# B&R Automation Studio project Teknologia25 (part 4)

#### Types.typ - Exported data types
```iecst
TYPE
	brfiShuttleSelectionType : 	STRUCT
		ID : DINT;
		index : DINT;
		x : REAL;
		y : REAL;
	END_STRUCT;
END_TYPE

(**)
(*----- brfi6DMoveQueue -----*)

TYPE
	brfi6DMoveQueueStateEnum :
		(
		brfi6DMOVEQUEUE_DISABLED,
		brfi6DMOVEQUEUE_RUN,
		brfi6DMOVEQUEUE_DONE,
		brfi6DMOVEQUEUE_ERROR
		);
	brfi6DMoveQueueFbType : 	STRUCT
		ShGetInfo : MC_BR_ShGetInfo_Acp6D;
		MoveInPlane : MC_BR_MoveInPlane_Acp6D;
		Move6D : MC_BR_Move6D_Acp6D;
		MoveArc : MC_BR_MoveArc_Acp6D;
		ShWaitTime : MC_BR_ShWaitTime_Acp6D;
		RotaryMotion : MC_BR_RotaryMotion_Acp6D;
		ShLevitation : MC_BR_ShLevitation_Acp6D;
		RotaryMotionSpin : MC_BR_RotaryMotionSpin_Acp6D;
		ShWaitCmdLb : MC_BR_ShWaitCmdLb_Acp6D;
	END_STRUCT;
	brfi6DMoveQueueIrnalType : 	STRUCT
		initialized : BOOL;
		onStateEntry : BOOL;
		lastState : brfi6DMoveQueueStateEnum;
		lastSubState : DINT;
		i : DINT;
		position : McAcp6DShPositionType;
		Xc : REAL;
		Yc : REAL;
		dx : REAL;
		dy : REAL;
		radius : REAL;
		angle : REAL;
	END_STRUCT;
	brfi6DMoveQueueActionsType : 	STRUCT
		acknowledge : BOOL;
		error : BOOL;
		done : BOOL;
		getInfo : BOOL;
	END_STRUCT;
	brfi6DMoveQueueExecuteType : 	STRUCT
		moveInPlane : BOOL;
		move6D : BOOL;
		moveArc : BOOL;
		wait : BOOL;
		moveRotary : BOOL;
		levitate : BOOL;
		spin : BOOL;
		readInfo : BOOL;
		waitCmdLb : BOOL;
	END_STRUCT;
	brfi6DMoveQueueCommandType : 	STRUCT
		mask : UINT;
		inPlane : McAcp6DInPlaneParType;
		inSpace : McAcp6DMove6DParType;
		moveMode6D : McAcp6DMoveModeEnum;
		waitTime : REAL;
		rotary : McAcp6DRotaryMotionParType;
		arc : McAcp6DArcParType;
		levitation : McAcp6DLevitationParType;
		spin : McAcp6DRotaryMotionSpinParType;
		waitCmdLb : brfi6DMoveWaitLabelParamType;
	END_STRUCT;
	brfi6DMoveQueueParamType : 	STRUCT
		velocity_xy : REAL;
		velocity_short : REAL;
		velocity_rotary : REAL;
		acceleration : REAL;
		acceleration_rotary : REAL;
	END_STRUCT;
	brfi6DMoveCommandSelectionEnum :
		(
		sX := 1,
		sY := 2,
		sZ := 4,
		sRx := 8,
		sRy := 16,
		sRz := 32,
		sArc := 64,
		sRotary := 128,
		sWait := 256,
		sLevitate := 512,
		sSpin := 1024,
		sUpdatePosition := 2048,
		sWaitCmdLb := 4096
		);
	brfi6DMoveCommandPathEnum :
		(
		pathDIRECT,
		pathX_Y,
		pathY_X
		);
	brfi6DMoveWaitLabelParamType : 	STRUCT
		monitoredShuttleID : UINT;
		triggerType : McAcp6DShWaitCmdLbTriggerEnum;
		commandLabel : UINT;
		labelType : McAcp6DShWaitCmdLbLabelEnum;
	END_STRUCT;
END_TYPE

(**)

TYPE
	Acp6dShuttleType : 	STRUCT  (*Global shuttle list datatype*)
		ID : UINT; (*ID of the shuttle*)
		Ref : Mc6DShuttleType; (*Reference to the shuttle*)
		index : DINT; (*ID of the shuttle*)
		status : Acp6dShuttleStatusType; (*Reference to the shuttle*)
		position : Acp6dShuttlePositionType;
		force : Acp6dShuttleForceType;
		command : Acp6dShuttleCmdType;
		moveCyclicActive : BOOL;
	END_STRUCT;
	Acp6dShuttleCmdType : 	STRUCT  (*Global shuttle list datatype*)
		move6D : BOOL; (*ID of the shuttle*)
		moveQueue : BOOL; (*ID of the shuttle*)
	END_STRUCT;
	Acp6dShuttlePositionType : 	STRUCT  (*Global shuttle list datatype*)
		isValid : BOOL; (*ID of the shuttle*)
		value : McAcp6DShPositionType; (*ID of the shuttle*)
	END_STRUCT;
	Acp6dShuttleForceType : 	STRUCT  (*Global shuttle list datatype*)
		isValid : BOOL; (*ID of the shuttle*)
		value : McAcp6DShForceType; (*ID of the shuttle*)
		Z_avg : REAL;
		Fz_baseline : REAL;
		readings : ARRAY[0..gMAX_INDEX_MEASUREMENT]OF McAcp6DShForceType;
	END_STRUCT;
	Acp6dShuttleStatusType : 	STRUCT  (*Global shuttle list datatype*)
		isValid : BOOL; (*ID of the shuttle*)
		state : McAcp6DShStateEnum; (*ID of the shuttle*)
	END_STRUCT;
END_TYPE

(**)

TYPE
	brfiShuttleGroupFbType : 	STRUCT
		GroupCreate : MC_BR_ShGroupCreate_Acp6D;
		GroupAddShuttle : MC_BR_ShGroupAddShuttle_Acp6D;
		GroupDelete : MC_BR_ShGroupDelete_Acp6D;
		GroupGetInfo : MC_BR_ShGroupGetInfo_Acp6D;
		GroupCoupleCtrl : MC_BR_ShGroupCoupleCtrl_Acp6D;
	END_STRUCT;
END_TYPE

(**)
```

#### Constants.var - Exported constants
```iecst
VAR CONSTANT
	MEASUREMENT_COUNT : DINT := 10;
	MAX_NUM_SHUTTLE : DINT := 8; (*Maximum numer of shuttles on the system*)
	MAX_NUM_SHUTTLE_VIRTUAL : DINT := 2; (*Maximum numer of shuttles on the system*)
	MAX_NUM_TARGETS : DINT := 20; (*Maximum numer of shuttles on the system*)
	SHUFFLE_SEQUENCE_LEN : DINT := 16;
END_VAR
(**)
VAR CONSTANT
	gMAX_INDEX_SHUTTLE : DINT := MAX_NUM_SHUTTLE - 1; (*Maximum index for a shuttles on the system*)
	gMAX_INDEX_SHUTTLE_VIRTUAL : DINT := MAX_NUM_SHUTTLE_VIRTUAL - 1; (*Maximum index for a shuttles on the system*)
	gMAX_INDEX_TARGETS : DINT := MAX_NUM_TARGETS - 1; (*Maximum index for a shuttles on the system*)
	gMAX_INDEX_MEASUREMENT : DINT := MEASUREMENT_COUNT - 1;
	gMAX_INDEX_SHUFFLE : DINT := SHUFFLE_SEQUENCE_LEN - 1;
END_VAR
(**)
```

#### brfiDemo.fun - Exported functions and function blocks
```iecst
{REDUND_ERROR} FUNCTION brfiShuffle : BOOL (* *) (*$GROUP=User,$CAT=User,$GROUPICON=User.png,$CATICON=User.png*)
	VAR_INPUT
		refArray : REFERENCE TO ARRAY[0..gMAX_INDEX_SHUTTLE] OF DINT;
	END_VAR
	VAR
		newOrder : ARRAY[0..gMAX_INDEX_SHUTTLE] OF DINT;
		added : ARRAY[0..gMAX_INDEX_SHUTTLE] OF BOOL;
		rand : DINT;
		count : DINT;
		i : DINT;
		ordinal : DINT;
		x : DINT;
	END_VAR
END_FUNCTION

FUNCTION brfiShuttleSelect : DINT
	VAR_INPUT
		Shuttles : REFERENCE TO ARRAY[0..gMAX_INDEX_SHUTTLE] OF Acp6dShuttleType;
		Selection : REFERENCE TO ARRAY[0..gMAX_INDEX_SHUTTLE] OF brfiShuttleSelectionType;
		X0 : REAL;
		Y0 : REAL;
		X1 : REAL;
		Y1 : REAL;
	END_VAR
	VAR
		i : DINT;
		j : DINT;
		count : DINT;
		maxX : REAL;
		maxY : REAL;
		minX : REAL;
		minY : REAL;
		key : brfiShuttleSelectionType;
	END_VAR
END_FUNCTION

FUNCTION brfiShuttleSelectClosest : DINT
	VAR_INPUT
		Shuttles : REFERENCE TO ARRAY[0..gMAX_INDEX_SHUTTLE] OF Acp6dShuttleType;
		X : REAL;
		Y : REAL;
	END_VAR
	VAR
		i : DINT;
		dist : REAL;
		dist_min : REAL;
		index_min : DINT;
	END_VAR
END_FUNCTION

FUNCTION brfiSortCompare : BOOL
	VAR_INPUT
		A : brfiShuttleSelectionType;
		B : brfiShuttleSelectionType;
		AscendingX : BOOL;
		AscendingY : BOOL;
	END_VAR
	VAR
		isEqualX : BOOL;
	END_VAR
END_FUNCTION

FUNCTION brfiToRAD : REAL
	VAR_INPUT
		degrees : REAL;
	END_VAR
END_FUNCTION

FUNCTION brfiToDEG : REAL
	VAR_INPUT
		radians : REAL;
	END_VAR
END_FUNCTION
(**)

{REDUND_ERROR} FUNCTION_BLOCK brfi6DMoveQueue (* *) (*$GROUP=User,$CAT=User,$GROUPICON=User.png,$CATICON=User.png*)
	VAR_INPUT
		Shuttle : REFERENCE TO Mc6DShuttleType;
		Execute : {REDUND_UNREPLICABLE} BOOL;
		Parameters : {REDUND_UNREPLICABLE} brfi6DMoveQueueParamType;
		Commands : {REDUND_UNREPLICABLE} ARRAY[0..gMAX_INDEX_TARGETS] OF brfi6DMoveQueueCommandType;
	END_VAR
	VAR_OUTPUT
		Done : {REDUND_UNREPLICABLE} BOOL;
		Acknowledge : {REDUND_UNREPLICABLE} BOOL;
		Error : {REDUND_UNREPLICABLE} BOOL;
		ErrorID : {REDUND_UNREPLICABLE} DINT;
		FailedCommand : {REDUND_UNREPLICABLE} brfi6DMoveQueueCommandType;
		FailedCommandIndex : {REDUND_UNREPLICABLE} DINT;
		LastExecutedState : {REDUND_UNREPLICABLE} DINT;
	END_VAR
	VAR
		refCommand : REFERENCE TO brfi6DMoveQueueCommandType;
		refAllCommandsDone : REFERENCE TO BOOL;
		state : {REDUND_UNREPLICABLE} brfi6DMoveQueueStateEnum;
		subState : {REDUND_UNREPLICABLE} DINT;
		onStateEntry : BOOL;
		fb : {REDUND_UNREPLICABLE} brfi6DMoveQueueFbType;
		actions : {REDUND_UNREPLICABLE} brfi6DMoveQueueActionsType;
		cmd : {REDUND_UNREPLICABLE} brfi6DMoveQueueExecuteType;
		internal : {REDUND_UNREPLICABLE} brfi6DMoveQueueIrnalType;
	END_VAR
END_FUNCTION_BLOCK

FUNCTION AddCommand6D_xy : BOOL
	VAR_INPUT
		Commands : REFERENCE TO ARRAY[0..gMAX_INDEX_TARGETS] OF brfi6DMoveQueueCommandType;
		axisSelect : brfi6DMoveCommandSelectionEnum;
		x : REAL;
		y : REAL;
		velocity : REAL;
		acceleration : REAL;
		endVelocity : REAL;
		path : brfi6DMoveCommandPathEnum;
		radius : REAL;
		mode : McAcp6DMoveModeEnum;
	END_VAR
	VAR
		i : DINT;
	END_VAR
END_FUNCTION

FUNCTION AddCommand6D_xyz : BOOL
	VAR_INPUT
		Commands : REFERENCE TO ARRAY[0..gMAX_INDEX_TARGETS] OF brfi6DMoveQueueCommandType;
		axisSelect : brfi6DMoveCommandSelectionEnum;
		x : REAL;
		y : REAL;
		z : REAL;
		velocity : REAL;
		velocity_short : REAL;
		acceleration : REAL;
		mode : McAcp6DMoveModeEnum;
	END_VAR
	VAR
		i : DINT;
	END_VAR
END_FUNCTION

FUNCTION AddCommand6D_Rxyz : BOOL
	VAR_INPUT
		Commands : REFERENCE TO ARRAY[0..gMAX_INDEX_TARGETS] OF brfi6DMoveQueueCommandType;
		axisSelect : brfi6DMoveCommandSelectionEnum;
		Rx : REAL;
		Ry : REAL;
		Rz : REAL;
		velocity_short : REAL;
		mode : McAcp6DMoveModeEnum;
	END_VAR
	VAR
		i : DINT;
	END_VAR
END_FUNCTION

FUNCTION AddCommand6D_wait : BOOL
	VAR_INPUT
		Commands : REFERENCE TO ARRAY[0..gMAX_INDEX_TARGETS] OF brfi6DMoveQueueCommandType;
		time : REAL; (*wait time in seconds*)
	END_VAR
	VAR
		i : DINT;
	END_VAR
END_FUNCTION

FUNCTION AddCommand6D_land : BOOL
	VAR_INPUT
		Commands : REFERENCE TO ARRAY[0..gMAX_INDEX_TARGETS] OF brfi6DMoveQueueCommandType;
		speed : USINT;
		Fz : REAL;
	END_VAR
	VAR
		i : DINT;
	END_VAR
END_FUNCTION

FUNCTION AddCommand6D_levitate : BOOL
	VAR_INPUT
		Commands : REFERENCE TO ARRAY[0..gMAX_INDEX_TARGETS] OF brfi6DMoveQueueCommandType;
		speed : USINT;
		Fz : REAL;
	END_VAR
	VAR
		i : DINT;
	END_VAR
END_FUNCTION

FUNCTION AddCommand6D_spin : BOOL
	VAR_INPUT
		Commands : REFERENCE TO ARRAY[0..gMAX_INDEX_TARGETS] OF brfi6DMoveQueueCommandType;
		duration : REAL; (*Duration of the rotational movement after reaching the target velocity (s)*)
		angle : REAL; (*Angle at which the shuttle stops after the rotational movement (rad)*)
		velocity : REAL; (*Rotational speed (rad/s)*)
		acceleration : REAL; (*Rotational acceleration (rad/s2)*)
	END_VAR
	VAR
		i : DINT;
	END_VAR
END_FUNCTION

FUNCTION AddCommand6D_rotateAbs : BOOL
	VAR_INPUT
		Commands : REFERENCE TO ARRAY[0..gMAX_INDEX_TARGETS] OF brfi6DMoveQueueCommandType;
		angle : REAL; (*Target angle (rad)*)
		velocity : REAL; (*Rotational speed (rad/s)*)
		acceleration : REAL; (*Rotational acceleration (rad/s2)*)
	END_VAR
	VAR
		i : DINT;
	END_VAR
END_FUNCTION

FUNCTION AddCommand6D_rotateCW : BOOL
	VAR_INPUT
		Commands : REFERENCE TO ARRAY[0..gMAX_INDEX_TARGETS] OF brfi6DMoveQueueCommandType;
		angle : REAL; (*Target angle (rad)*)
		velocity : REAL; (*Rotational speed (rad/s)*)
		acceleration : REAL; (*Rotational acceleration (rad/s2)*)
	END_VAR
	VAR
		i : DINT;
	END_VAR
END_FUNCTION

FUNCTION AddCommand6D_rotateCCW : BOOL
	VAR_INPUT
		Commands : REFERENCE TO ARRAY[0..gMAX_INDEX_TARGETS] OF brfi6DMoveQueueCommandType;
		angle : REAL; (*Target angle (rad)*)
		velocity : REAL; (*Rotational speed (rad/s)*)
		acceleration : REAL; (*Rotational acceleration (rad/s2)*)
	END_VAR
	VAR
		i : DINT;
	END_VAR
END_FUNCTION

FUNCTION AddCommand6D_arcAngularCW : BOOL
	VAR_INPUT
		Commands : REFERENCE TO ARRAY[0..gMAX_INDEX_TARGETS] OF brfi6DMoveQueueCommandType;
		x : REAL;
		y : REAL;
		angle : REAL;
		velocity : REAL;
		acceleration : REAL;
		endVelocity : REAL;
		mode : McAcp6DMoveModeEnum;
	END_VAR
	VAR
		i : DINT;
	END_VAR
END_FUNCTION

FUNCTION AddCommand6D_arcAngularCCW : BOOL
	VAR_INPUT
		Commands : REFERENCE TO ARRAY[0..gMAX_INDEX_TARGETS] OF brfi6DMoveQueueCommandType;
		x : REAL;
		y : REAL;
		angle : REAL;
		velocity : REAL;
		acceleration : REAL;
		endVelocity : REAL;
		mode : McAcp6DMoveModeEnum;
	END_VAR
	VAR
		i : DINT;
	END_VAR
END_FUNCTION

FUNCTION AddCommand6D_arcRadialCW : BOOL
	VAR_INPUT
		Commands : REFERENCE TO ARRAY[0..gMAX_INDEX_TARGETS] OF brfi6DMoveQueueCommandType;
		x : REAL;
		y : REAL;
		radius : REAL;
		type : McAcp6DArcTypeEnum; (*Rotational speed (rad/s)*)
		velocity : REAL; (*Rotational speed (rad/s)*)
		acceleration : REAL; (*Rotational acceleration (rad/s2)*)
		endVelocity : REAL; (*Target angle (rad)*)
		mode : McAcp6DMoveModeEnum;
	END_VAR
	VAR
		i : DINT;
	END_VAR
END_FUNCTION

FUNCTION AddCommand6D_arcRadialCCW : BOOL
	VAR_INPUT
		Commands : REFERENCE TO ARRAY[0..gMAX_INDEX_TARGETS] OF brfi6DMoveQueueCommandType;
		x : REAL;
		y : REAL;
		radius : REAL;
		type : McAcp6DArcTypeEnum; (*Rotational speed (rad/s)*)
		velocity : REAL; (*Rotational speed (rad/s)*)
		acceleration : REAL; (*Rotational acceleration (rad/s2)*)
		endVelocity : REAL; (*Target angle (rad)*)
		mode : McAcp6DMoveModeEnum;
	END_VAR
	VAR
		i : DINT;
	END_VAR
END_FUNCTION

FUNCTION AddCommand6D_waitCmdLb : BOOL
	VAR_INPUT
		Commands : REFERENCE TO ARRAY[0..gMAX_INDEX_TARGETS] OF brfi6DMoveQueueCommandType;
		monitoredShuttleID : UINT;
		triggerType : McAcp6DShWaitCmdLbTriggerEnum;
		commandLabel : UINT;
		labelType : McAcp6DShWaitCmdLbLabelEnum;
	END_VAR
	VAR
		i : DINT;
	END_VAR
END_FUNCTION
(**)

{REDUND_ERROR} FUNCTION_BLOCK brfiShuttleGroup (* *) (*$GROUP=User,$CAT=User,$GROUPICON=User.png,$CATICON=User.png*)
	VAR_INPUT
		Assembly : REFERENCE TO Mc6DAssemblyType;
		Shuttles : {REDUND_UNREPLICABLE} ARRAY[0..gMAX_INDEX_SHUTTLE] OF Mc6DShuttleType;
		Enable : {REDUND_UNREPLICABLE} BOOL;
	END_VAR
	VAR_OUTPUT
		Inactive : {REDUND_UNREPLICABLE} BOOL;
		Active : {REDUND_UNREPLICABLE} BOOL;
		Busy : {REDUND_UNREPLICABLE} BOOL;
		Error : {REDUND_UNREPLICABLE} BOOL;
		ErrorID : {REDUND_UNREPLICABLE} DINT;
		NumberOfShuttles : {REDUND_UNREPLICABLE} UINT;
	END_VAR
	VAR
		shuttleGroupRef : Mc6DShuttleGroupType;
		state : {REDUND_UNREPLICABLE} DINT;
		i : {REDUND_UNREPLICABLE} DINT;
		fb : {REDUND_UNREPLICABLE} brfiShuttleGroupFbType;
	END_VAR
END_FUNCTION_BLOCK
(**)

{REDUND_ERROR} FUNCTION_BLOCK brfiSunPlanet (* *) (*$GROUP=User,$CAT=User,$GROUPICON=User.png,$CATICON=User.png*)
	VAR_INPUT
		SunShuttle : REFERENCE TO Mc6DShuttleType;
		PlanetShuttles : {REDUND_UNREPLICABLE} ARRAY[0..gMAX_INDEX_SHUTTLE] OF Mc6DShuttleType;
		Enable : {REDUND_UNREPLICABLE} BOOL;
	END_VAR
	VAR_OUTPUT
		Active : {REDUND_UNREPLICABLE} BOOL;
		Busy : {REDUND_UNREPLICABLE} BOOL;
		Error : {REDUND_UNREPLICABLE} BOOL;
		ErrorID : {REDUND_UNREPLICABLE} DINT;
	END_VAR
	VAR
		state : {REDUND_UNREPLICABLE} DINT;
		i : {REDUND_UNREPLICABLE} DINT;
		ShPlanet : {REDUND_UNREPLICABLE} MC_BR_ShPlanet_Acp6D;
	END_VAR
END_FUNCTION_BLOCK
```

#### Common.st
```iecst
(*  *)
FUNCTION brfiShuffle

	count := gMAX_INDEX_SHUTTLE;

	FOR i := 0 TO gMAX_INDEX_SHUTTLE DO
		rand := RandValueDINT(0, count);
		ordinal := 0;

		FOR x := 0 TO gMAX_INDEX_SHUTTLE DO
			IF NOT added[x] THEN
				ordinal := ordinal + 1;
			END_IF;

			IF (rand + 1) = ordinal THEN
				EXIT;
			END_IF;
		END_FOR;

		added[x] := TRUE;
		newOrder[x] := refArray[i];
		count := count - 1;

	END_FOR;

	brsmemcpy(ADR(refArray), ADR(newOrder), SIZEOF(refArray));

END_FUNCTION

FUNCTION brfiShuttleSelect

	// First find shuttles that are in the selection area
	maxX := MAX(X0, X1);
	maxY := MAX(Y0, Y1);
	minX := MIN(X0, X1);
	minY := MIN(Y0, Y1);
	brsmemset(ADR(Selection), 0, SIZEOF(Selection));

	FOR i := 0 TO gMAX_INDEX_SHUTTLE DO
		IF Shuttles[i].position.value.X < maxX AND Shuttles[i].position.value.X > minX THEN
			IF Shuttles[i].position.value.Y < maxY AND Shuttles[i].position.value.Y > minY THEN
				Selection[count].index := Shuttles[i].index;
				Selection[count].ID := Shuttles[i].ID;
				Selection[count].x := Shuttles[i].position.value.X;
				Selection[count].y := Shuttles[i].position.value.Y;
				count := count + 1;
			END_IF;
		END_IF;
	END_FOR;

	brfiShuttleSelect := count;

	IF count < 2 THEN
		RETURN;
	END_IF;

	// Sort selection array by X
	FOR i := 1 TO count - 1 DO
		key := Selection[i];
		j := i - 1;

		// Compare key with each element on the LEFT OF it UNTIL an element smaller than it is found
		WHILE j >= 0 AND brfiSortCompare(key, Selection[j], (X0 < X1), (Y0 < Y1)) DO
			Selection[j + 1] := Selection[j];
			j := j - 1;
			Selection[j + 1] := key;
		END_WHILE;
	END_FOR

END_FUNCTION

FUNCTION brfiShuttleSelectClosest

	dist_min := 1000000;

	FOR i := 0 TO gMAX_INDEX_SHUTTLE DO
		dist := SQRT(EXPT(X - Shuttles[i].position.value.X, 2) + EXPT(Y - Shuttles[i].position.value.Y, 2));

		IF  dist < dist_min THEN
			dist_min := dist;
	  		index_min := i;
		END_IF;
	END_FOR;

	brfiShuttleSelectClosest := index_min;

END_FUNCTION

FUNCTION brfiSortCompare
	// Comparison function for two pairs (A, B)

	IF AscendingX THEN
		// X needs to be sorted in ascending order
		IF A.x < B.x THEN
			brfiSortCompare := TRUE;
			RETURN;
		END_IF;
	ELSE
		// X needs to be sorted in descending order
		IF A.x > B.x THEN
			brfiSortCompare := TRUE;
			RETURN;
		END_IF;
	END_IF;

	isEqualX := ABS(A.x - B.x) < 0.001;

	IF isEqualX THEN
		// Only sort by Y if X is equal as we primarily sort by X
		IF AscendingY THEN
			// Y needs to be sorted in ascending order
			IF A.y < B.y THEN
				brfiSortCompare := TRUE;
				RETURN;
			END_IF;
		ELSE
			// Y needs to be sorted in descending order
			IF A.y > B.y THEN
				brfiSortCompare := TRUE;
				RETURN;
			END_IF;
		END_IF;
	END_IF;

END_FUNCTION

FUNCTION brfiToRAD

	brfiToRAD := degrees * brmPI / 180.0;

END_FUNCTION

FUNCTION brfiToDEG

	brfiToDEG := radians / brmPI * 180.0;

END_FUNCTION
```

#### MoveQueue.st
```iecst
FUNCTION_BLOCK brfi6DMoveQueue

    // Execution control
    // ========================================================================================================
	IF Execute = FALSE THEN
		IF internal.initialized THEN
			brsmemset(ADR(internal), 0, SIZEOF(internal));
			brsmemset(ADR(actions), 0, SIZEOF(actions));
		END_IF
		state := brfi6DMOVEQUEUE_DISABLED;
	END_IF

	// Program code
	// ========================================================================================================
	CASE state OF
		brfi6DMOVEQUEUE_DISABLED:
			//
			// ------------------------------------------------------
			IF Execute THEN
				internal.initialized := TRUE;
				brsmemset(ADR(FailedCommand), 0, SIZEOF(FailedCommand));
				brsmemset(ADR(cmd), 0, SIZEOF(cmd));
				FailedCommandIndex := -1;
				ErrorID := 0;
				state := brfi6DMOVEQUEUE_RUN;
			END_IF;

		brfi6DMOVEQUEUE_RUN:
			CASE subState OF
				0:
					// ------------------------------------------------------
					actions.getInfo := TRUE;

					IF fb.ShGetInfo.Done THEN
						internal.position := fb.ShGetInfo.ShuttleInfo.Position;
						subState := 100;
					ELSIF fb.ShGetInfo.Error THEN
						ErrorID := fb.ShGetInfo.ErrorID;
						state := brfi6DMOVEQUEUE_ERROR;
					END_IF;

				100:
					// Find next target that has masked axes
					// ------------------------------------------------------
					IF internal.i > gMAX_INDEX_TARGETS THEN
						state := brfi6DMOVEQUEUE_DONE;
					END_IF;

					WHILE internal.i <= gMAX_INDEX_TARGETS DO
						refCommand ACCESS ADR(Commands[internal.i]);

						IF refCommand.mask > 0 THEN
							// Select movement type based on the AxisMask for the target
							IF refCommand.mask <= 3 THEN
								cmd.moveInPlane := FALSE;
								subState := 200;
	  						ELSIF refCommand.mask <= 32 THEN
								cmd.move6D := FALSE;
								subState := 300;
							ELSIF refCommand.mask = sArc THEN
								cmd.moveArc := FALSE;
								subState := 400;
							ELSIF refCommand.mask = sRotary THEN
								cmd.moveRotary := FALSE;
								subState := 500;
							ELSIF refCommand.mask = sWait THEN
								cmd.wait := FALSE;
								subState := 600;
							ELSIF refCommand.mask = sLevitate THEN
								cmd.levitate := FALSE;
								subState := 700;
							ELSIF refCommand.mask = sSpin THEN
								cmd.spin := FALSE;
								subState := 800;
							ELSIF refCommand.mask = sWaitCmdLb THEN
								cmd.waitCmdLb := FALSE;
								subState := 900;
							ELSE
								state := brfi6DMOVEQUEUE_ERROR;
								ErrorID := 666;
								FailedCommand := refCommand;
							END_IF;

							internal.i := internal.i + 1;
							EXIT;
						END_IF;

						internal.i := internal.i + 1;
					END_WHILE;

				200:
					// ------------------------------------------------------------------------------------------------------------
					IF onStateEntry THEN
	  					brsmemset(ADR(fb.MoveInPlane.Parameters), 0, SIZEOF(fb.MoveInPlane.Parameters));

						// Use target velocity/acceleration when available. Use values from parameters as fallback values
						fb.MoveInPlane.Parameters.Velocity := SEL(refCommand.inPlane.Velocity > 0, Parameters.velocity_xy, refCommand.inPlane.Velocity);
						fb.MoveInPlane.Parameters.Acceleration := SEL(refCommand.inPlane.Acceleration > 0, Parameters.acceleration, refCommand.inPlane.Acceleration);
						fb.MoveInPlane.Parameters.EndVelocity := refCommand.inPlane.EndVelocity;

						fb.MoveInPlane.Parameters.Path := refCommand.inPlane.Path;
						fb.MoveInPlane.Parameters.Radius := refCommand.inPlane.Radius;
						fb.MoveInPlane.Parameters.Mode := refCommand.inPlane.Mode;

						IF refCommand.inPlane.Mode = mcACP6D_MOVE_ABSOLUTE THEN
							fb.MoveInPlane.Parameters.Position.X := SEL(refCommand.mask.0, internal.position.X, refCommand.inPlane.Position.X);
							fb.MoveInPlane.Parameters.Position.Y := SEL(refCommand.mask.1, internal.position.Y, refCommand.inPlane.Position.Y);

							// Update shuttles current position for next command
							internal.position.X := fb.MoveInPlane.Parameters.Position.X;
							internal.position.Y := fb.MoveInPlane.Parameters.Position.Y;
						ELSE
							fb.MoveInPlane.Parameters.Position.X := SEL(refCommand.mask.0, 0, refCommand.inPlane.Position.X);
							fb.MoveInPlane.Parameters.Position.Y := SEL(refCommand.mask.1, 0, refCommand.inPlane.Position.Y);

							// Update shuttles current position for next command
							internal.position.X := internal.position.X + fb.MoveInPlane.Parameters.Position.X;
							internal.position.Y := internal.position.Y + fb.MoveInPlane.Parameters.Position.Y;
						END_IF;
					END_IF;

					cmd.moveInPlane := TRUE;

					IF fb.MoveInPlane.Acknowledge THEN
						refAllCommandsDone ACCESS ADR(fb.MoveInPlane.Done);
						subState := 100;
					ELSIF fb.MoveInPlane.Error THEN
						ErrorID := fb.MoveInPlane.ErrorID;
						FailedCommand.inPlane := fb.MoveInPlane.Parameters;
						state := brfi6DMOVEQUEUE_ERROR;
					END_IF;

				300:
					// ------------------------------------------------------------------------------------------------------------
					IF onStateEntry THEN

						brsmemset(ADR(fb.Move6D.Parameters), 0, SIZEOF(fb.Move6D.Parameters));
						fb.Move6D.Parameters := refCommand.inSpace;

						// Use target velocity/acceleration when available. Use values from parameters as fallback values
						IF fb.Move6D.Parameters.InPlane.Velocity = 0 THEN fb.Move6D.Parameters.InPlane.Velocity := Parameters.velocity_xy; END_IF;
						IF fb.Move6D.Parameters.InPlane.Acceleration = 0 THEN fb.Move6D.Parameters.InPlane.Acceleration := Parameters.acceleration; END_IF;

						IF fb.Move6D.Parameters.ShortAxis.Velocity.Z = 0 THEN fb.Move6D.Parameters.ShortAxis.Velocity.Z := Parameters.velocity_short; END_IF;
						IF fb.Move6D.Parameters.ShortAxis.Velocity.Rx = 0 THEN fb.Move6D.Parameters.ShortAxis.Velocity.Rx := Parameters.velocity_short; END_IF;
						IF fb.Move6D.Parameters.ShortAxis.Velocity.Ry = 0 THEN fb.Move6D.Parameters.ShortAxis.Velocity.Ry := Parameters.velocity_short; END_IF;
						IF fb.Move6D.Parameters.ShortAxis.Velocity.Rz = 0 THEN fb.Move6D.Parameters.ShortAxis.Velocity.Rz := Parameters.velocity_short; END_IF;

						IF refCommand.moveMode6D = mcACP6D_MOVE_ABSOLUTE THEN
							// Set absolute target
							fb.Move6D.Parameters.InPlane.Position.X := SEL(refCommand.mask.0,  internal.position.X, refCommand.inSpace.InPlane.Position.X);
							fb.Move6D.Parameters.InPlane.Position.Y := SEL(refCommand.mask.1,  internal.position.Y, refCommand.inSpace.InPlane.Position.Y);
							fb.Move6D.Parameters.ShortAxis.Position.Z := SEL(refCommand.mask.2,  internal.position.Z, refCommand.inSpace.ShortAxis.Position.Z);
							fb.Move6D.Parameters.ShortAxis.Position.Rx := SEL(refCommand.mask.3,  internal.position.Rx, refCommand.inSpace.ShortAxis.Position.Rx);
							fb.Move6D.Parameters.ShortAxis.Position.Ry := SEL(refCommand.mask.4,  internal.position.Ry, refCommand.inSpace.ShortAxis.Position.Ry);
							fb.Move6D.Parameters.ShortAxis.Position.Rz := SEL(refCommand.mask.5,  internal.position.Rz, refCommand.inSpace.ShortAxis.Position.Rz);
						END_IF

						IF refCommand.moveMode6D = mcACP6D_MOVE_RELATIVE THEN
							// Calculate relative target
							fb.Move6D.Parameters.InPlane.Position.X := SEL(refCommand.mask.0,  internal.position.X, internal.position.X + refCommand.inSpace.InPlane.Position.X);
							fb.Move6D.Parameters.InPlane.Position.Y := SEL(refCommand.mask.1,  internal.position.Y, internal.position.Y + refCommand.inSpace.InPlane.Position.Y);
							fb.Move6D.Parameters.ShortAxis.Position.Z := SEL(refCommand.mask.2,  internal.position.Z, internal.position.Z + refCommand.inSpace.ShortAxis.Position.Z);
							fb.Move6D.Parameters.ShortAxis.Position.Rx := SEL(refCommand.mask.3,  internal.position.Rx, internal.position.Rx + refCommand.inSpace.ShortAxis.Position.Rx);
							fb.Move6D.Parameters.ShortAxis.Position.Ry := SEL(refCommand.mask.4,  internal.position.Ry, internal.position.Ry + refCommand.inSpace.ShortAxis.Position.Ry);
							fb.Move6D.Parameters.ShortAxis.Position.Rz := SEL(refCommand.mask.5,  internal.position.Rz, internal.position.Rz + refCommand.inSpace.ShortAxis.Position.Rz);
						END_IF;

						// Update current shuttle position based on latest move command. 6D move moves always naturally to absolute
						// positions so we can just set the parameter positions as our current position now
						internal.position.X := fb.Move6D.Parameters.InPlane.Position.X;
						internal.position.Y := fb.Move6D.Parameters.InPlane.Position.Y;
						internal.position.Z := fb.Move6D.Parameters.ShortAxis.Position.Z;
						internal.position.Rx := fb.Move6D.Parameters.ShortAxis.Position.Rx;
						internal.position.Ry := fb.Move6D.Parameters.ShortAxis.Position.Ry;
						internal.position.Rz := fb.Move6D.Parameters.ShortAxis.Position.Rz;
					END_IF;

					cmd.move6D := TRUE;

					IF fb.Move6D.Acknowledge THEN
						refAllCommandsDone ACCESS ADR(fb.Move6D.Done);
						subState := 100;
					ELSIF fb.Move6D.Error THEN
						ErrorID := fb.Move6D.ErrorID;
						FailedCommand.inSpace := fb.Move6D.Parameters;
						state := brfi6DMOVEQUEUE_ERROR;
					END_IF;

				400:
					// ------------------------------------------------------------------------------------------------------------
					IF onStateEntry THEN
						fb.MoveArc.Parameters := refCommand.arc;
						fb.MoveArc.Parameters.Velocity := SEL(refCommand.arc.Velocity > 0, Parameters.velocity_xy, refCommand.arc.Velocity);
						fb.MoveArc.Parameters.Acceleration := SEL(refCommand.arc.Acceleration > 0, Parameters.acceleration, refCommand.arc.Acceleration);

						// Radius move mode
						IF fb.MoveArc.Parameters.Option = mcACP6D_ARC_RADIUS THEN
							IF fb.MoveArc.Parameters.Mode = mcACP6D_MOVE_ABSOLUTE THEN
								internal.position.X := fb.MoveArc.Parameters.Radius.Position.X;
								internal.position.Y := fb.MoveArc.Parameters.Radius.Position.Y;
							END_IF

							IF fb.MoveArc.Parameters.Mode = mcACP6D_MOVE_RELATIVE THEN
								internal.position.X := internal.position.X + fb.MoveArc.Parameters.Radius.Position.X;
								internal.position.Y := internal.position.Y + fb.MoveArc.Parameters.Radius.Position.Y;
							END_IF
						END_IF

						// Angular move mode
						IF fb.MoveArc.Parameters.Option = mcACP6D_ARC_ANGULAR THEN
							IF fb.MoveArc.Parameters.Mode = mcACP6D_MOVE_ABSOLUTE THEN
								internal.Xc := fb.MoveArc.Parameters.Angular.Center.X;
								internal.Yc := fb.MoveArc.Parameters.Angular.Center.Y;
							END_IF

							IF fb.MoveArc.Parameters.Mode = mcACP6D_MOVE_RELATIVE THEN
								internal.Xc := internal.position.X + fb.MoveArc.Parameters.Angular.Center.X;
								internal.Yc := internal.position.Y + fb.MoveArc.Parameters.Angular.Center.Y;
							END_IF
						END_IF

						internal.dx := internal.position.X - internal.Xc;
						internal.dy := internal.position.Y - internal.Yc;

						// Calculate end position after arc move
						internal.radius := SQRT(EXPT(internal.position.X - internal.Xc, 2) + EXPT(internal.position.Y - internal.Yc, 2));
						internal.angle := brmatan2(internal.dy, internal.dx);

						// Natural rotation direction for trigonometric functions is CCW so if we are
						// moving CW then we need to invert the angle value before summing
						IF fb.MoveArc.Parameters.Direction = mcACP6D_ARC_COUNTER_CLOCKWISE THEN
							internal.angle := internal.angle + fb.MoveArc.Parameters.Angular.Angle;
						ELSE
	  						internal.angle := internal.angle - fb.MoveArc.Parameters.Angular.Angle;
						END_IF;

						internal.position.X := internal.Xc + internal.radius * COS(internal.angle);
						internal.position.Y := internal.Yc + internal.radius * SIN(internal.angle);
					END_IF

					cmd.moveArc := TRUE;

					IF fb.MoveArc.Acknowledge THEN
						refAllCommandsDone ACCESS ADR(fb.MoveArc.Done);
						subState := 100;
					ELSIF fb.MoveArc.Error THEN
						ErrorID := fb.MoveArc.ErrorID;
						FailedCommand.arc := fb.MoveArc.Parameters;
						state := brfi6DMOVEQUEUE_ERROR;
					END_IF;

				500:
					// ------------------------------------------------------------------------------------------------------------
					IF onStateEntry THEN
						fb.RotaryMotion.Parameters := refCommand.rotary;
						fb.RotaryMotion.Parameters.Velocity := SEL(refCommand.rotary.Velocity > 0, Parameters.velocity_rotary, refCommand.rotary.Velocity);
						fb.RotaryMotion.Parameters.Acceleration := SEL(refCommand.rotary.Acceleration > 0, Parameters.acceleration_rotary, refCommand.rotary.Acceleration);
					END_IF;

					cmd.moveRotary := TRUE;

					IF fb.RotaryMotion.Acknowledge THEN
						refAllCommandsDone ACCESS ADR(fb.RotaryMotion.Done);
						subState := 100;
					ELSIF fb.RotaryMotion.Error THEN
						ErrorID := fb.RotaryMotion.ErrorID;
						FailedCommand.rotary := fb.RotaryMotion.Parameters;
						state := brfi6DMOVEQUEUE_ERROR;
					END_IF;

				600:
					// ------------------------------------------------------------------------------------------------------------
					IF onStateEntry THEN
						fb.ShWaitTime.Delay := refCommand.waitTime;
					END_IF;

					cmd.wait := TRUE;

					IF fb.ShWaitTime.Acknowledge THEN
						refAllCommandsDone ACCESS ADR(fb.ShWaitTime.Done);
						subState := 100;
					ELSIF fb.ShWaitTime.Error THEN
						ErrorID := fb.ShWaitTime.ErrorID;
						FailedCommand.waitTime := fb.ShWaitTime.Delay;
						state := brfi6DMOVEQUEUE_ERROR;
					END_IF;

				700:
					// ------------------------------------------------------------------------------------------------------------
					IF onStateEntry THEN
						fb.ShLevitation.Parameters := refCommand.levitation;
					END_IF;

					cmd.levitate := TRUE;

					IF fb.ShLevitation.Acknowledge THEN
						refAllCommandsDone ACCESS ADR(fb.ShLevitation.Done);
						subState := 100;
					ELSIF fb.ShLevitation.Error THEN
						ErrorID := fb.ShLevitation.ErrorID;
						FailedCommand.levitation := fb.ShLevitation.Parameters;
						state := brfi6DMOVEQUEUE_ERROR;
					END_IF;

				800:
					// ------------------------------------------------------------------------------------------------------------
					IF onStateEntry THEN
						fb.RotaryMotionSpin.Parameters := refCommand.spin;
						fb.RotaryMotionSpin.Parameters.Velocity := SEL(refCommand.spin.Velocity > 0, Parameters.velocity_rotary, refCommand.spin.Velocity);
						fb.RotaryMotionSpin.Parameters.Acceleration := SEL(refCommand.spin.Acceleration > 0, Parameters.acceleration_rotary, refCommand.spin.Acceleration);
					END_IF;

					cmd.spin := TRUE;

					IF fb.RotaryMotionSpin.Acknowledge THEN
						refAllCommandsDone ACCESS ADR(fb.RotaryMotionSpin.Done);
						subState := 100;
					ELSIF fb.RotaryMotionSpin.Error THEN
						ErrorID := fb.RotaryMotionSpin.ErrorID;
						FailedCommand.spin := fb.RotaryMotionSpin.Parameters;
						state := brfi6DMOVEQUEUE_ERROR;
					END_IF;

				900:
					// ------------------------------------------------------------------------------------------------------------
					IF onStateEntry THEN
						fb.ShWaitCmdLb.TriggerXID := refCommand.waitCmdLb.monitoredShuttleID;
						fb.ShWaitCmdLb.CommandLabel := refCommand.waitCmdLb.commandLabel;
						fb.ShWaitCmdLb.LabelType := refCommand.waitCmdLb.labelType;
						fb.ShWaitCmdLb.TriggerType := refCommand.waitCmdLb.triggerType;
					END_IF;

					cmd.waitCmdLb := TRUE;

					IF fb.ShWaitCmdLb.Acknowledge THEN
						refAllCommandsDone ACCESS ADR(fb.ShWaitCmdLb.Done);
						subState := 100;
					ELSIF fb.ShWaitCmdLb.Error THEN
						ErrorID := fb.ShWaitCmdLb.ErrorID;
						FailedCommand.waitCmdLb := refCommand.waitCmdLb;
						state := brfi6DMOVEQUEUE_ERROR;
					END_IF;
			END_CASE;

		brfi6DMOVEQUEUE_DONE:
			//
			// ------------------------------------------------------
			actions.acknowledge := TRUE;

			// If pointer is not set then just indicate all done as this means queue contained
			// no valid commands and nothing was queued to 6D controller.
			// Otherwise wait for the last called function block to finish to indicate shuttles has
			// executed all of its queued commands
			IF ADR(refAllCommandsDone) = 0 THEN
				actions.done := TRUE;
			ELSE
				actions.done := refAllCommandsDone;
			END_IF;

		brfi6DMOVEQUEUE_ERROR:
			//
			// ------------------------------------------------------
			FailedCommandIndex := internal.i - 1;
			actions.error := TRUE;

	END_CASE;

	// State change events
	// -------------------------------------------------------------------
	onStateEntry := (state <> internal.lastState) OR (subState <> internal.lastSubState);

	IF state <> internal.lastState THEN
		subState := 0;
		brsmemset(ADR(actions), 0, SIZEOF(actions));
		internal.lastState := state;
	END_IF;

	// Reset current state actions also when substate changes
	IF subState <> internal.lastSubState THEN
		internal.lastSubState := subState;
		LastExecutedState := internal.lastSubState;
		brsmemset(ADR(actions), 0, SIZEOF(actions));
	END_IF

	// Function calls
	// ========================================================================================================
	fb.ShGetInfo.Shuttle := ADR(Shuttle);
	fb.ShGetInfo.Execute := actions.getInfo;
	fb.ShGetInfo();

	fb.MoveInPlane.Shuttle := ADR(Shuttle);
	fb.MoveInPlane.Execute := cmd.moveInPlane;
	fb.MoveInPlane();

	fb.Move6D.Shuttle := ADR(Shuttle);
	fb.Move6D.Execute := cmd.move6D;
	fb.Move6D();

	fb.MoveArc.Shuttle := ADR(Shuttle);
	fb.MoveArc.Execute := cmd.moveArc;
	fb.MoveArc();

	fb.RotaryMotion.Shuttle := ADR(Shuttle);
	fb.RotaryMotion.Execute := cmd.moveRotary;
	fb.RotaryMotion();

	fb.ShWaitTime.Shuttle := ADR(Shuttle);
	fb.ShWaitTime.Execute := cmd.wait;
	fb.ShWaitTime();

	fb.ShLevitation.Shuttle := ADR(Shuttle);
	fb.ShLevitation.Execute := cmd.levitate;
	fb.ShLevitation();

	fb.RotaryMotionSpin.Shuttle := ADR(Shuttle);
	fb.RotaryMotionSpin.Execute := cmd.spin;
	fb.RotaryMotionSpin();

	fb.ShWaitCmdLb.Shuttle := ADR(Shuttle);
	fb.ShWaitCmdLb.Execute := cmd.waitCmdLb;
	fb.ShWaitCmdLb();

	// Outputs
	// ========================================================================================================
	Done := actions.done;
	Acknowledge := actions.acknowledge;
	Error := actions.error;

END_FUNCTION_BLOCK
```

#### AddCommand6D.st
```iecst
// XY plane move
// ========================================================================================================
FUNCTION AddCommand6D_xy
	FOR i := 0 TO gMAX_INDEX_TARGETS DO
		IF Commands[i].mask = 0 THEN
			Commands[i].mask := DINT_TO_UINT(axisSelect);
			Commands[i].inPlane.Position.X := x;
			Commands[i].inPlane.Position.Y := y;
			Commands[i].inPlane.Velocity := velocity;
			Commands[i].inPlane.EndVelocity := endVelocity;
			Commands[i].inPlane.Acceleration := acceleration;
			Commands[i].inPlane.Radius := radius;
			Commands[i].inPlane.Mode := mode;

			CASE path OF
				pathDIRECT:
					Commands[i].inPlane.Path := mcACP6D_PATH_DIRECT;
				pathX_Y:
					Commands[i].inPlane.Path := mcACP6D_PATH_X_THEN_Y;
				pathY_X:
		  			Commands[i].inPlane.Path := mcACP6D_PATH_Y_THEN_X;
			END_CASE;

			AddCommand6D_xy := TRUE;
			RETURN;
		END_IF;
	END_FOR;
END_FUNCTION

// 6D move
// ========================================================================================================
FUNCTION AddCommand6D_xyz
	FOR i := 0 TO gMAX_INDEX_TARGETS DO
		IF Commands[i].mask = 0 THEN
			Commands[i].mask := DINT_TO_UINT(axisSelect);
			Commands[i].inSpace.InPlane.Position.X := x;
			Commands[i].inSpace.InPlane.Position.Y := y;
			Commands[i].inSpace.ShortAxis.Position.Z := z;
			Commands[i].inSpace.InPlane.Velocity := velocity;
			Commands[i].inSpace.InPlane.Acceleration := acceleration;
			Commands[i].inSpace.ShortAxis.Velocity.Z := velocity_short;
			Commands[i].moveMode6D := mode;
			AddCommand6D_xyz := TRUE;
			RETURN;
		END_IF;
	END_FOR;
END_FUNCTION

FUNCTION AddCommand6D_Rxyz
	FOR i := 0 TO gMAX_INDEX_TARGETS DO
		IF Commands[i].mask = 0 THEN
			Commands[i].mask := DINT_TO_UINT(axisSelect);
			Commands[i].inSpace.ShortAxis.Position.Rx := Rx;
			Commands[i].inSpace.ShortAxis.Position.Ry := Ry;
			Commands[i].inSpace.ShortAxis.Position.Rz := Rz;
			Commands[i].inSpace.ShortAxis.Velocity.Z := velocity_short;
			Commands[i].inSpace.ShortAxis.Velocity.Rx := velocity_short;
			Commands[i].inSpace.ShortAxis.Velocity.Ry := velocity_short;
			Commands[i].inSpace.ShortAxis.Velocity.Rz := velocity_short;
			Commands[i].moveMode6D := mode;
			AddCommand6D_Rxyz := TRUE;
			RETURN;
		END_IF;
	END_FOR;
END_FUNCTION

// Wait
// ========================================================================================================
FUNCTION AddCommand6D_wait
	FOR i := 0 TO gMAX_INDEX_TARGETS DO
		IF Commands[i].mask = 0 THEN
			Commands[i].mask := DINT_TO_UINT(sWait);
			Commands[i].waitTime := time;
			AddCommand6D_wait := TRUE;
			RETURN;
		END_IF;
	END_FOR;
END_FUNCTION

FUNCTION AddCommand6D_waitCmdLb
	FOR i := 0 TO gMAX_INDEX_TARGETS DO
		IF Commands[i].mask = 0 THEN
			Commands[i].mask := DINT_TO_UINT(sWaitCmdLb);
			Commands[i].waitCmdLb.monitoredShuttleID := monitoredShuttleID;
			Commands[i].waitCmdLb.triggerType := triggerType;
			Commands[i].waitCmdLb.commandLabel := commandLabel;
			Commands[i].waitCmdLb.labelType := labelType;
			AddCommand6D_waitCmdLb := TRUE;
			RETURN;
		END_IF;
	END_FOR;
END_FUNCTION

// Rotary
// ========================================================================================================
FUNCTION AddCommand6D_rotateAbs
	FOR i := 0 TO gMAX_INDEX_TARGETS DO
		IF Commands[i].mask = 0 THEN
			Commands[i].mask := DINT_TO_UINT(sRotary);
			Commands[i].rotary.Angle := angle;
			Commands[i].rotary.Velocity := velocity;
			Commands[i].rotary.Acceleration := acceleration;
			Commands[i].rotary.Mode := mcACP6D_ROTATE_ABSOLUTE_POS;
			AddCommand6D_rotateAbs := TRUE;
			RETURN;
		END_IF;
	END_FOR;
END_FUNCTION

FUNCTION AddCommand6D_rotateCW
	FOR i := 0 TO gMAX_INDEX_TARGETS DO
		IF Commands[i].mask = 0 THEN
			Commands[i].mask := DINT_TO_UINT(sRotary);
			Commands[i].rotary.Angle := angle;
			Commands[i].rotary.Velocity := velocity;
			Commands[i].rotary.Acceleration := acceleration;
			Commands[i].rotary.Mode := mcACP6D_ROTATE_CLOCKWISE;
			AddCommand6D_rotateCW := TRUE;
			RETURN;
		END_IF;
	END_FOR;
END_FUNCTION

FUNCTION AddCommand6D_rotateCCW
	FOR i := 0 TO gMAX_INDEX_TARGETS DO
		IF Commands[i].mask = 0 THEN
			Commands[i].mask := DINT_TO_UINT(sRotary);
			Commands[i].rotary.Angle := angle;
			Commands[i].rotary.Velocity := velocity;
			Commands[i].rotary.Acceleration := acceleration;
			Commands[i].rotary.Mode := mcACP6D_ROTATE_COUNTER_CLOCKWISE;
			AddCommand6D_rotateCCW := TRUE;
			RETURN;
		END_IF;
	END_FOR;
END_FUNCTION

// Arc
// ========================================================================================================
FUNCTION AddCommand6D_arcAngularCW
	FOR i := 0 TO gMAX_INDEX_TARGETS DO
		IF Commands[i].mask = 0 THEN
			Commands[i].mask := DINT_TO_UINT(sArc);
			Commands[i].arc.Velocity := velocity;
			Commands[i].arc.EndVelocity := endVelocity;
			Commands[i].arc.Acceleration := acceleration;
			Commands[i].arc.Angular.Angle := angle;
			Commands[i].arc.Angular.Center.X := x;
			Commands[i].arc.Angular.Center.Y := y;
			Commands[i].arc.Mode := mode;
			Commands[i].arc.Direction := mcACP6D_ARC_CLOCKWISE;
			Commands[i].arc.Option := mcACP6D_ARC_ANGULAR;
			AddCommand6D_arcAngularCW := TRUE;
			RETURN;
		END_IF;
	END_FOR;
END_FUNCTION

FUNCTION AddCommand6D_arcAngularCCW
	FOR i := 0 TO gMAX_INDEX_TARGETS DO
		IF Commands[i].mask = 0 THEN
			Commands[i].mask := DINT_TO_UINT(sArc);
			Commands[i].arc.Velocity := velocity;
			Commands[i].arc.EndVelocity := endVelocity;
			Commands[i].arc.Acceleration := acceleration;
			Commands[i].arc.Angular.Angle := angle;
			Commands[i].arc.Angular.Center.X := x;
			Commands[i].arc.Angular.Center.Y := y;
			Commands[i].arc.Mode := mode;
			Commands[i].arc.Direction := mcACP6D_ARC_COUNTER_CLOCKWISE;
			Commands[i].arc.Option := mcACP6D_ARC_ANGULAR;
			AddCommand6D_arcAngularCCW := TRUE;
			RETURN;
		END_IF;
	END_FOR;
END_FUNCTION

FUNCTION AddCommand6D_arcRadialCW
	FOR i := 0 TO gMAX_INDEX_TARGETS DO
		IF Commands[i].mask = 0 THEN
			Commands[i].mask := DINT_TO_UINT(sArc);
			Commands[i].arc.Velocity := velocity;
			Commands[i].arc.EndVelocity := endVelocity;
			Commands[i].arc.Acceleration := acceleration;
			Commands[i].arc.Radius.Position.X := x;
			Commands[i].arc.Radius.Position.Y := y;
			Commands[i].arc.Radius.Radius := radius;
			Commands[i].arc.Radius.ArcType := type;
			Commands[i].arc.Mode := mode;
			Commands[i].arc.Direction := mcACP6D_ARC_CLOCKWISE;
			Commands[i].arc.Option := mcACP6D_ARC_RADIUS;
			AddCommand6D_arcRadialCW := TRUE;
			RETURN;
		END_IF;
	END_FOR;
END_FUNCTION

FUNCTION AddCommand6D_arcRadialCCW
	FOR i := 0 TO gMAX_INDEX_TARGETS DO
		IF Commands[i].mask = 0 THEN
			Commands[i].mask := DINT_TO_UINT(sArc);
			Commands[i].arc.Velocity := velocity;
			Commands[i].arc.EndVelocity := endVelocity;
			Commands[i].arc.Acceleration := acceleration;
			Commands[i].arc.Radius.Position.X := x;
			Commands[i].arc.Radius.Position.Y := y;
			Commands[i].arc.Radius.Radius := radius;
			Commands[i].arc.Radius.ArcType := type;
			Commands[i].arc.Mode := mode;
			Commands[i].arc.Direction := mcACP6D_ARC_COUNTER_CLOCKWISE;
			Commands[i].arc.Option := mcACP6D_ARC_RADIUS;
			AddCommand6D_arcRadialCCW := TRUE;
			RETURN;
		END_IF;
	END_FOR;
END_FUNCTION

// Spin
// ========================================================================================================
FUNCTION AddCommand6D_spin
	FOR i := 0 TO gMAX_INDEX_TARGETS DO
		IF Commands[i].mask = 0 THEN
			Commands[i].mask := DINT_TO_UINT(sSpin);
			Commands[i].spin.Duration := duration;
			Commands[i].spin.Angle := angle;
			Commands[i].spin.Velocity := velocity;
			Commands[i].spin.Acceleration := acceleration;
			AddCommand6D_spin := TRUE;
			RETURN;
		END_IF;
	END_FOR;
END_FUNCTION

// Levitation
// ========================================================================================================
FUNCTION AddCommand6D_levitate
	FOR i := 0 TO gMAX_INDEX_TARGETS DO
		IF Commands[i].mask = 0 THEN
			Commands[i].mask := DINT_TO_UINT(sLevitate);
			Commands[i].levitation.Level := mcACP6D_LEVEL_LEVITATE;
			Commands[i].levitation.Speed := speed;
			Commands[i].levitation.ZForce := Fz;
			AddCommand6D_levitate := TRUE;
			RETURN;
		END_IF;
	END_FOR;
END_FUNCTION

FUNCTION AddCommand6D_land
	FOR i := 0 TO gMAX_INDEX_TARGETS DO
		IF Commands[i].mask = 0 THEN
			Commands[i].mask := DINT_TO_UINT(sLevitate);
			Commands[i].levitation.Level := mcACP6D_LEVEL_LAND;
			Commands[i].levitation.Speed := speed;
			Commands[i].levitation.ZForce := Fz;
			AddCommand6D_land := TRUE;
			RETURN;
		END_IF;
	END_FOR;
END_FUNCTION
```

#### ShuttleGroup.st
```iecst
FUNCTION_BLOCK brfiShuttleGroup

	fb.GroupAddShuttle.Execute := FALSE;
	fb.GroupCreate.Execute := FALSE;
	fb.GroupDelete.Execute := FALSE;
	fb.GroupGetInfo.Execute := FALSE;
	fb.GroupCoupleCtrl.Execute := FALSE;

	Active := FALSE;
	Error := FALSE;
	Inactive := FALSE;

	// Program code
	// ========================================================================================================
	CASE state OF
		0:
			// Inactive
			// -------------------------------------------------------------------
			Inactive := TRUE;
			ErrorID := 0;
			NumberOfShuttles := 0;

			IF Enable THEN
				state := 10;
			END_IF;

		10:
			// Create group
			// -------------------------------------------------------------------
			fb.GroupCreate.Execute := TRUE;

			IF fb.GroupCreate.Done THEN
				shuttleGroupRef := fb.GroupCreate.ShuttleGroup;
				state := 20;
			ELSIF fb.GroupCreate.Error THEN
				ErrorID := fb.GroupCreate.ErrorID;
	  			state := 100;
			END_IF;

		20:
			// Add shuttles to the group
			// -------------------------------------------------------------------
			brsmemset(ADR(fb.GroupAddShuttle.Parameters), 0, SIZEOF(fb.GroupAddShuttle.Parameters));

			FOR i := 0 TO gMAX_INDEX_SHUTTLE DO
				IF Shuttles[i].controlif > 0 THEN
	  				fb.GroupAddShuttle.Parameters.ShuttleList[i].Shuttle := ADR(Shuttles[i]);
				END_IF;
			END_FOR;

			fb.GroupAddShuttle.Execute := TRUE;

			IF fb.GroupCreate.Done THEN
				state := 30;
			ELSIF fb.GroupCreate.Error THEN
				ErrorID := fb.GroupCreate.ErrorID;
				state := 100;
			END_IF;

		30:
			// Read group info
			// -------------------------------------------------------------------
			fb.GroupGetInfo.Execute := TRUE;

			IF fb.GroupGetInfo.Done THEN
				NumberOfShuttles := fb.GroupGetInfo.Info.NumberOfShuttles;
				state := 40;
			ELSIF fb.GroupGetInfo.Error THEN
				ErrorID := fb.GroupGetInfo.ErrorID;
				state := 100;
			END_IF;

		40:
			// Couple shuttles together
			// -------------------------------------------------------------------
			fb.GroupCoupleCtrl.Parameters.Mode :=  mcACP6D_SH_GROUP_INDV_ROT_REF;
			fb.GroupCoupleCtrl.Parameters.Option := mcACP6D_SH_GROUP_COUPLE;

			fb.GroupCoupleCtrl.Execute := TRUE;

			IF fb.GroupCoupleCtrl.Done THEN
				state := 50;
			ELSIF fb.GroupCoupleCtrl.Error THEN
				ErrorID := fb.GroupGetInfo.ErrorID;
				state := 100;
			END_IF;

		50:
			// Group active
			// -------------------------------------------------------------------
			Active := TRUE;

			IF NOT Enable THEN
				state := 60;
			END_IF;

		60:
			// Delete group
			// -------------------------------------------------------------------
			fb.GroupDelete.Execute := TRUE;

			IF fb.GroupDelete.Done THEN
				state := 0;
			ELSIF fb.GroupDelete.Error THEN
				ErrorID := fb.GroupCreate.ErrorID;
				state := 100;
			END_IF;

		100:
			// -------------------------------------------------------------------
			Error := TRUE;

			IF NOT Enable THEN
	  			state := 0;
			END_IF;
	END_CASE;

	// Function calls
	// ========================================================================================================
	fb.GroupCreate.Assembly := ADR(Assembly);
	fb.GroupCreate();

	fb.GroupAddShuttle.ShuttleGroup := ADR(shuttleGroupRef);
	fb.GroupAddShuttle();

	fb.GroupDelete.ShuttleGroup :=  ADR(shuttleGroupRef);
	fb.GroupDelete();

	fb.GroupGetInfo.ShuttleGroup :=  ADR(shuttleGroupRef);
	fb.GroupGetInfo();

	fb.GroupCoupleCtrl.ShuttleGroup :=  ADR(shuttleGroupRef);
	fb.GroupCoupleCtrl();

	Busy := fb.GroupCreate.Busy OR fb.GroupAddShuttle.Busy OR fb.GroupDelete.Busy OR fb.GroupGetInfo.Busy;

END_FUNCTION_BLOCK
```

#### SunPlanet.st
```iecst
FUNCTION_BLOCK brfiSunPlanet

	ShPlanet.Execute := FALSE;

	Active := FALSE;
	Error := FALSE;

	// Program code
	// ========================================================================================================
	CASE state OF
		0:
			// Inactive
			// -------------------------------------------------------------------
			ErrorID := 0;

			IF Enable THEN
				state := 10;
			END_IF;

		10:
			// Create sun planet system
			// -------------------------------------------------------------------
			ShPlanet.Execute := TRUE;
			ShPlanet.Parameters.Option := mcACP6D_PLANET_ADD_SH;

			ShPlanet.Shuttle := ADR(SunShuttle);

			brsmemset(ADR(ShPlanet.Parameters.ShuttleList), 0, SIZEOF(ShPlanet.Parameters.ShuttleList));

			FOR i := 0 TO gMAX_INDEX_SHUTTLE DO
				IF PlanetShuttles[i].controlif > 0 THEN
					ShPlanet.Parameters.ShuttleList[i].Shuttle := ADR(PlanetShuttles[i]);
				END_IF;
			END_FOR;

			IF ShPlanet.Done THEN
				state := 20;
			ELSIF ShPlanet.Error THEN
				ErrorID := ShPlanet.ErrorID;
	  			state := 100;
			END_IF;

		20:
			// Sun planet system active and coupled
			// -------------------------------------------------------------------
			Active := TRUE;

			IF NOT Enable THEN
	  			state := 30;
			END_IF;

		30:
			// Decouple sun planet system
			// -------------------------------------------------------------------
			ShPlanet.Execute := TRUE;
			ShPlanet.Parameters.Option := mcACP6D_PLANET_REMOVE_SH;

			IF ShPlanet.Done THEN
				state := 0;
			ELSIF ShPlanet.Error THEN
				ErrorID := ShPlanet.ErrorID;
				state := 100;
			END_IF;

		100:
			// -------------------------------------------------------------------
			Error := TRUE;

			IF NOT Enable THEN
				state := 0;
			END_IF;
	END_CASE;

	// Function calls
	// ========================================================================================================
	ShPlanet();

	Busy := ShPlanet.Busy;

END_FUNCTION_BLOCK
```

#### Move6DQueue.st - not listed in the package file held
```iecst
(*  *)
FUNCTION AddTarget6D_xyz

	FOR i := 0 TO gMAX_INDEX_TARGETS DO
		IF TargetList[i].axisMask = 0 THEN
			TargetList[i].axisMask := DINT_TO_USINT(axisSelect);
			TargetList[i].x := x;
			TargetList[i].y := y;
			TargetList[i].z := z;
			TargetList[i].velocity_xy := velocity_xy;
			TargetList[i].velocity_short := velocity_short;
			TargetList[i].acceleration := acceleration;
			TargetList[i].mode := mode;
			RETURN;
		END_IF;
	END_FOR;

END_FUNCTION

FUNCTION AddTarget6D_Rxyz

	FOR i := 0 TO gMAX_INDEX_TARGETS DO
		IF TargetList[i].axisMask = 0 THEN
			TargetList[i].axisMask := DINT_TO_USINT(axisSelect);
			TargetList[i].Rx := Rx;
			TargetList[i].Ry := Ry;
			TargetList[i].Rz := Rz;
			TargetList[i].velocity_short := velocity_short;
			TargetList[i].mode := mode;
			RETURN;
		END_IF;
	END_FOR;

END_FUNCTION

FUNCTION AddTarget6D_all

	FOR i := 0 TO gMAX_INDEX_TARGETS DO
		IF TargetList[i].axisMask = 0 THEN
			TargetList[i].axisMask := DINT_TO_USINT(axisSelect);
			TargetList[i].x := x;
			TargetList[i].y := y;
			TargetList[i].z := z;
			TargetList[i].Rx := Rx;
			TargetList[i].Ry := Ry;
			TargetList[i].Rz := Rz;
			TargetList[i].velocity_xy := velocity_xy;
			TargetList[i].velocity_short := velocity_short;
			TargetList[i].acceleration := acceleration;
			TargetList[i].mode := mode;
			RETURN;
		END_IF;
	END_FOR;

END_FUNCTION

FUNCTION_BLOCK brfiMove6DQueue

    // Execution control
    // ========================================================================================================
	IF Execute = FALSE THEN
		IF internal.initialized THEN
			brsmemset(ADR(internal), 0, SIZEOF(internal));
		END_IF
		state := brfiMOVE6DQUEUE_DISABLED;
	END_IF

	// Program code
	// ========================================================================================================
	CASE state OF
		brfiMOVE6DQUEUE_DISABLED:
			//
			// ------------------------------------------------------
			Move6D.Execute := FALSE;

			IF Execute THEN
				internal.initialized := TRUE;
				state := brfiMOVE6DQUEUE_RUN;
			END_IF;

		brfiMOVE6DQUEUE_RUN:
			CASE subState OF
				0:
					// Read current position of the shuttle
					// ------------------------------------------------------
					internal.actions.executeReadPosition := TRUE;

					IF ShGetInfo.Done THEN
						internal.position := ShGetInfo.ShuttleInfo.Position;
						subState := 10;
					ELSIF ShGetInfo.Error THEN
						LastStatusCode := ShGetInfo.ErrorID;
						state := brfiMOVE6DQUEUE_ERROR;
					END_IF;

				10:
					// Find next target that has masked axes
					// ------------------------------------------------------
					IF internal.i > gMAX_INDEX_TARGETS THEN
						state := brfiMOVE6DQUEUE_DONE;
					END_IF;

					WHILE internal.i <= gMAX_INDEX_TARGETS DO
						refTarget ACCESS ADR(Targets[internal.i]);

						IF refTarget.axisMask > 0 THEN
							internal.i := internal.i + 1;
							Move6D.Execute := FALSE;
							brsmemset(ADR(Move6D.Parameters), 0, SIZEOF(Move6D.Parameters));

							// Use target velocity/acceleration when available. Use values from parameters as fallback values
							Move6D.Parameters.InPlane.Velocity := SEL(refTarget.velocity_xy > 0, Parameters.velocity_xy, refTarget.velocity_xy);
							Move6D.Parameters.InPlane.Acceleration := SEL(refTarget.acceleration > 0, Parameters.acceleration, refTarget.acceleration);

							IF refTarget.velocity_short > 0 THEN
								Move6D.Parameters.ShortAxis.Velocity.Z := refTarget.velocity_short;
								Move6D.Parameters.ShortAxis.Velocity.Rx := refTarget.velocity_short;
								Move6D.Parameters.ShortAxis.Velocity.Ry := refTarget.velocity_short;
								Move6D.Parameters.ShortAxis.Velocity.Rz := refTarget.velocity_short;
							ELSE
								Move6D.Parameters.ShortAxis.Velocity.Z := Parameters.velocity_short;
								Move6D.Parameters.ShortAxis.Velocity.Rx := Parameters.velocity_short;
								Move6D.Parameters.ShortAxis.Velocity.Ry := Parameters.velocity_short;
								Move6D.Parameters.ShortAxis.Velocity.Rz := Parameters.velocity_short;
							END_IF;

							IF refTarget.mode = brfiMOVE6D_ABSOLUTE THEN
								// Set absolute target
								Move6D.Parameters.InPlane.Position.X := SEL(refTarget.axisMask.0,  internal.position.X, refTarget.x);
								Move6D.Parameters.InPlane.Position.Y := SEL(refTarget.axisMask.1,  internal.position.Y, refTarget.y);
								Move6D.Parameters.ShortAxis.Position.Z := SEL(refTarget.axisMask.2,  internal.position.Z, refTarget.z);
								Move6D.Parameters.ShortAxis.Position.Rx := SEL(refTarget.axisMask.3,  internal.position.Rx, refTarget.Rx);
								Move6D.Parameters.ShortAxis.Position.Ry := SEL(refTarget.axisMask.4,  internal.position.Ry, refTarget.Ry);
								Move6D.Parameters.ShortAxis.Position.Rz := SEL(refTarget.axisMask.5,  internal.position.Rz, refTarget.Rz);
							ELSE
								// Calculate relative target
								Move6D.Parameters.InPlane.Position.X := SEL(refTarget.axisMask.0,  internal.position.X, internal.position.X + refTarget.x);
								Move6D.Parameters.InPlane.Position.Y := SEL(refTarget.axisMask.1,  internal.position.Y, internal.position.Y + refTarget.y);
								Move6D.Parameters.ShortAxis.Position.Z := SEL(refTarget.axisMask.2,  internal.position.Z, internal.position.Z + refTarget.z);
								Move6D.Parameters.ShortAxis.Position.Rx := SEL(refTarget.axisMask.3,  internal.position.Rx, internal.position.Rx + refTarget.Rx);
								Move6D.Parameters.ShortAxis.Position.Ry := SEL(refTarget.axisMask.4,  internal.position.Ry, internal.position.Ry + refTarget.Ry);
								Move6D.Parameters.ShortAxis.Position.Rz := SEL(refTarget.axisMask.5,  internal.position.Rz, internal.position.Rz + refTarget.Rz);
							END_IF;
							subState := 20;
							EXIT;
						END_IF;

						internal.i := internal.i + 1;
					END_WHILE;

				20:
					// Add to queue
					// ------------------------------------------------------
					Move6D.Execute := TRUE;

					IF Move6D.Acknowledge THEN
						// Update current position with the target we just added to the command queue
						internal.position.X := Move6D.Parameters.InPlane.Position.X;
						internal.position.Y := Move6D.Parameters.InPlane.Position.Y;
						internal.position.Z := Move6D.Parameters.ShortAxis.Position.Z;
						internal.position.Rx := Move6D.Parameters.ShortAxis.Position.Rx;
						internal.position.Ry := Move6D.Parameters.ShortAxis.Position.Ry;
						internal.position.Rz := Move6D.Parameters.ShortAxis.Position.Rz;
						subState := 10;
					ELSIF Move6D.Error THEN
						LastStatusCode := Move6D.ErrorID;
						state := brfiMOVE6DQUEUE_ERROR;
					END_IF;
			END_CASE;

		brfiMOVE6DQUEUE_DONE:
			//
			// ------------------------------------------------------
			internal.actions.ready := TRUE;

		brfiMOVE6DQUEUE_ERROR:
			//
			// ------------------------------------------------------
			Move6D.Execute := FALSE;
			internal.actions.error := TRUE;

	END_CASE;

	// State change events
	// -------------------------------------------------------------------
	IF state <> internal.lastState THEN
		// If function block is enabled -> update info of last executed state
		IF Execute THEN
			LastExecutedState := internal.lastState;
		END_IF;

		subState := 0;
		brsmemset(ADR(internal.actions), 0, SIZEOF(internal.actions));
		internal.lastState := state;
	END_IF;

	// Reset current state actions also when substate changes
	IF subState <> internal.lastSubState THEN
		internal.lastSubState := subState;
		brsmemset(ADR(internal.actions), 0, SIZEOF(internal.actions));
	END_IF

	// Function calls
	// ========================================================================================================
	Move6D.Shuttle := ADR(Shuttle);
	Move6D();

	ShGetInfo.Shuttle := ADR(Shuttle);
	ShGetInfo.Execute := internal.actions.executeReadPosition;
	ShGetInfo();

	// Outputs
	// ========================================================================================================
	Done := Move6D.Done;
	Ready := internal.actions.ready;
	Error := internal.actions.error;

END_FUNCTION_BLOCK
```

#### MoveXYQueue.st - not listed in the package file held
```iecst
FUNCTION AddTargetDIR

	FOR i := 0 TO gMAX_INDEX_TARGETS DO
		IF TargetList[i].axisMask = 0 THEN
			TargetList[i].axisMask := DINT_TO_USINT(axisSelect);
			TargetList[i].x := x;
			TargetList[i].y := y;
			TargetList[i].velocity := velocity;
			TargetList[i].acceleration := acceleration;
			TargetList[i].mode := mode;
			TargetList[i].path := mcACP6D_PATH_DIRECT;
			TargetList[i].radius := radius;
			RETURN;
		END_IF;
	END_FOR;

END_FUNCTION

FUNCTION AddTargetYX

	FOR i := 0 TO gMAX_INDEX_TARGETS DO
		IF TargetList[i].axisMask = 0 THEN
			TargetList[i].axisMask := DINT_TO_USINT(axisSelect);
			TargetList[i].x := x;
			TargetList[i].y := y;
			TargetList[i].velocity := velocity;
			TargetList[i].acceleration := acceleration;
			TargetList[i].mode := mode;
			TargetList[i].path := mcACP6D_PATH_Y_THEN_X;
			TargetList[i].radius := radius;
			RETURN;
		END_IF;
	END_FOR;

END_FUNCTION

FUNCTION AddTargetXY

	FOR i := 0 TO gMAX_INDEX_TARGETS DO
		IF TargetList[i].axisMask = 0 THEN
			TargetList[i].axisMask := DINT_TO_USINT(axisSelect);
			TargetList[i].x := x;
			TargetList[i].y := y;
			TargetList[i].velocity := velocity;
			TargetList[i].acceleration := acceleration;
			TargetList[i].mode := mode;
			TargetList[i].path := mcACP6D_PATH_X_THEN_Y;
			TargetList[i].radius := radius;
			RETURN;
		END_IF;
	END_FOR;

END_FUNCTION

FUNCTION_BLOCK brfiMoveXYQueue

    // Execution control
    // ========================================================================================================
	IF Execute = FALSE THEN
		IF internal.initialized THEN
			brsmemset(ADR(internal), 0, SIZEOF(internal));
		END_IF
		state := brfiMOVEXYQUEUE_DISABLED;
	END_IF

	// Program code
	// ========================================================================================================
	CASE state OF
		brfiMOVEXYQUEUE_DISABLED:
			//
			// ------------------------------------------------------
			MoveXY.Execute := FALSE;

			IF Execute THEN
				internal.initialized := TRUE;
				state := brfiMOVEXYQUEUE_RUN;
			END_IF;

		brfiMOVEXYQUEUE_RUN:
			CASE subState OF
				0:
					// ------------------------------------------------------
					internal.actions.executeReadPosition := TRUE;

					IF ShGetInfo.Done THEN
						internal.position.X := ShGetInfo.ShuttleInfo.Position.X;
						internal.position.Y := ShGetInfo.ShuttleInfo.Position.Y;
						subState := 10;
					ELSIF ShGetInfo.Error THEN
						LastStatusCode := ShGetInfo.ErrorID;
						state := brfiMOVEXYQUEUE_ERROR;
					END_IF;

				10:
					// Find next target that has masked axes
					// ------------------------------------------------------
					IF internal.i > gMAX_INDEX_TARGETS THEN
						state := brfiMOVEXYQUEUE_DONE;
					END_IF;

					WHILE internal.i <= gMAX_INDEX_TARGETS DO
						refTarget ACCESS ADR(Targets[internal.i]);

						IF (refTarget.axisMask > 0) OR (refTarget.mode = mcACP6D_MOVE_RELATIVE) THEN
							internal.i := internal.i + 1;
							MoveXY.Execute := FALSE;
							brsmemset(ADR(MoveXY.Parameters), 0, SIZEOF(MoveXY.Parameters));

							// Use target velocity/acceleration when available. Use values from parameters as fallback values
							MoveXY.Parameters.Velocity := SEL(refTarget.velocity > 0, Parameters.velocity, refTarget.velocity);
							MoveXY.Parameters.Acceleration := SEL(refTarget.acceleration > 0, Parameters.acceleration, refTarget.acceleration);
							MoveXY.Parameters.Path := refTarget.path;
							MoveXY.Parameters.Radius := refTarget.radius;
							MoveXY.Parameters.Mode := refTarget.mode;

							IF refTarget.mode = mcACP6D_MOVE_RELATIVE THEN
								MoveXY.Parameters.Position.X := refTarget.x;
								MoveXY.Parameters.Position.Y := refTarget.y;
							ELSE
								MoveXY.Parameters.Position.X := SEL(refTarget.axisMask.0, internal.position.X, refTarget.x);
								MoveXY.Parameters.Position.Y := SEL(refTarget.axisMask.1, internal.position.Y, refTarget.y);
							END_IF;

							MoveXY.Parameters.EndVelocity := 0;

							subState := 20;
							EXIT;
						END_IF;

						internal.i := internal.i + 1;
					END_WHILE;

				20:
					// Add to queue
					// ------------------------------------------------------
					MoveXY.Execute := TRUE;

					IF MoveXY.Acknowledge THEN
						// Update current shuttle position
						IF refTarget.mode = mcACP6D_MOVE_RELATIVE THEN
							internal.position.X := internal.position.X + MoveXY.Parameters.Position.X;
							internal.position.Y := internal.position.Y + MoveXY.Parameters.Position.Y;
						ELSE
							internal.position.X := MoveXY.Parameters.Position.X;
							internal.position.Y := MoveXY.Parameters.Position.Y;
						END_IF;

						subState := 10;
					ELSIF MoveXY.Error THEN
						LastStatusCode := MoveXY.ErrorID;
						state := brfiMOVEXYQUEUE_ERROR;
					END_IF;
			END_CASE;

		brfiMOVEXYQUEUE_DONE:
			//
			// ------------------------------------------------------
			internal.actions.ready := TRUE;

		brfiMOVEXYQUEUE_ERROR:
			//
			// ------------------------------------------------------
			MoveXY.Execute := FALSE;
			internal.actions.error := TRUE;

	END_CASE;

	// State change events
	// -------------------------------------------------------------------
	IF state <> internal.lastState THEN
		// If function block is enabled -> update info of last executed state
		IF Execute THEN
			LastExecutedState := internal.lastState;
		END_IF;

		subState := 0;
		brsmemset(ADR(internal.actions), 0, SIZEOF(internal.actions));
		internal.lastState := state;
	END_IF;

	// Reset current state actions also when substate changes
	IF subState <> internal.lastSubState THEN
		internal.lastSubState := subState;
		brsmemset(ADR(internal.actions), 0, SIZEOF(internal.actions));
	END_IF

	// Function calls
	// ========================================================================================================
	MoveXY.Shuttle := ADR(Shuttle);
	MoveXY();

	ShGetInfo.Shuttle := ADR(Shuttle);
	ShGetInfo.Execute := internal.actions.executeReadPosition;
	ShGetInfo();

	// Outputs
	// ========================================================================================================
	Done := MoveXY.Done;
	Ready := internal.actions.ready;
	Error := internal.actions.error;

END_FUNCTION_BLOCK
```

### global.var
```iecst
VAR
    gAcp6D : Acp6DType := (0);
END_VAR
```

### global.typ
```iecst
(*
Program: Acp6D

Description
(short summary)

*)
(*========== STATES ==========*)

TYPE
	Acp6DStateEnum :
		(
		ACP6D_INITIALIZE,
		ACP6D_IDLE,
		ACP6D_MOVE_TO,
		ACP6D_ERROR,
		ACP6D_COMMAND_ERROR,
		ACP6D_COMMAND_DONE,
		ACP6D_SELECT_SHUTTLE,
		ACP6D_FIND_PAYLOAD,
		ACP6D_SHUFFLE_SIMPLE,
		ACP6D_SHUFFLE_CIRCULAR,
		ACP6D_STOP_ALL,
		ACP6D_FORCE_RESET,
		ACP6D_VICTORY,
		ACP6D_ANIMATE,
		ACP6D_DEMO
		);
END_TYPE

(*========== INPUTS ==========*)

TYPE
	Acp6DInputCommandType : 	STRUCT
		Reinitialize : BOOL;
		ForceReset : BOOL;
		StopAll : BOOL;
		Victory : BOOL;
		Animate : BOOL;
		MoveTo : Acp6DMoveToCommandType;
		FindPayload : BOOL;
		SelectShuttle : BOOL;
		Shuffle : Acp6DShuffleCommandType;
		StartDemoMode : BOOL;
		StopDemoMode : BOOL;
	END_STRUCT;
	Acp6DMoveToCommandType : 	STRUCT
		Home : BOOL;
		User : BOOL;
		Pickup : BOOL;
		Shuffle : BOOL;
		Clockface : BOOL;
		Dance : BOOL;
		Side : BOOL;
	END_STRUCT;
	Acp6DShuffleCommandType : 	STRUCT
		Simple : BOOL;
		Circular : BOOL;
	END_STRUCT;
	Acp6DInputStatusType : 	STRUCT
		test : BOOL;
	END_STRUCT;
	Acp6DInputType : 	STRUCT
		Force : BOOL;
		Command : Acp6DInputCommandType;
		Status : Acp6DInputStatusType;
	END_STRUCT;
END_TYPE

(*========== OUTPUTS ==========*)

TYPE
	Acp6DOutputStatusType : 	STRUCT
		Initialized : BOOL;
		CommandDone : BOOL;
		DemoModeActive : BOOL;
	END_STRUCT;
	Acp6DOutputType : 	STRUCT
		Status : Acp6DOutputStatusType;
		TotalShuttleCount : DINT;
		AssemblyInfo : McAcp6DAsmInfoType;
		ShuttleWithPayload : Acp6DOutputShuttleType;
		ShuttleUserSelected : Acp6DOutputShuttleType;
	END_STRUCT;
	Acp6DOutputShuttleType : 	STRUCT
		index : DINT;
		X : REAL;
		Y : REAL;
	END_STRUCT;
END_TYPE

(*========== ERRORS ==========*)

TYPE
	Acp6DErrorType : 	STRUCT
		Active : BOOL;
		Acknowledge : BOOL;
		Code : DINT;
		State : Acp6DStateEnum;
		SubState : DINT;
	END_STRUCT;
END_TYPE

(*========== INTERFACE ==========*)

TYPE
	Acp6DType : 	STRUCT
		Error : Acp6DErrorType;
		Input : Acp6DInputType;
		Output : Acp6DOutputType;
		IsSimulated : BOOL;
		State : Acp6DStateEnum;
		SubState : DINT;
		StateInfo : STRING[255];
		OnStateEntry : BOOL; (*True for one cycle after state change*)
	END_STRUCT;
END_TYPE
```

### Program Logical/Acp6D/Acp6D (IEC)
